TYPE WcStateInputToggleBase_F68C23A9 :
STRUCT
END_STRUCT
END_TYPE

(* stored: Version 1.2.0.0, ProductVersion 3.1.4024.9
   DUT WcStateInputToggleBase_F68C23A9: Id {c835d4d8-1294-46cc-9df6-89526abae21a} *)
